Fanuc KAREL source: kt00186.KL

-- PROVISIONAL review KL for V1013-1; original PC SHA256 fb5a126682b29e7667c3fe8208325c7c00bd43973aaacdbc47d44d2b4d76703a
-- Incomplete behavior may be omitted. Consult companion uncertainty JSON. Do not deploy.
PROGRAM KT00186
%NOLOCKGROUP
VAR
  I2 : INTEGER
  OUT : REAL
-- UNRESOLVED_DECL H1 type=002017
BEGIN
  -- UNRESOLVED_PC offsets 5-19; opcodes 2E,22,9D,33,B4
  -- UNRESOLVED_PC offsets 24-35; opcodes 2E,23
  -- UNRESOLVED_PC offsets 40-63; opcodes 22,9D,33,B3,21,56,64,23
  -- UNRESOLVED_PC offsets 68-72; opcodes 7F
END KT00186
